{attribute 'qualified_only'}
VAR_GLOBAL
	bSwitchs AT%I* : ARRAY[1..8] OF BOOL;
	bLamps   AT%Q* : ARRAY[1..4] OF BOOL;

END_VAR

(* stored: Version 1.1.0.1, ProductVersion 3.1.4024.12
   GVL GVL_IO: Id {3c6bf2cb-4f4a-446c-965c-fbcb57f48134} *)
